// TIA Portal  export
FUNCTION_BLOCK "MissingVersion_FB"   // FB, LAD
// stored: SetENOAutomatically false
BEGIN
END_FUNCTION_BLOCK
